Omron Sysmac Studio project 3.0_integration_v3 (Sysmac Studio 1.54.0.64019, StandardProject)

# Controller new_Controller_0: NJ301-1100 version 1.14
Units and slaves: Node1 : NX-ECC201 (E001); Unit 1 : NX-PC0020 (N1); Unit 2 : NX-ID5442 (N2); Unit 3 : NX-PC0010 (N3); Unit 4 : NX-PC0020 (N4); Unit 5 : NX-OD5121 (N5); Unit 6 : NX-PC0010 (N6); Power Supply : NJ-Px3001; CPU : NJ301-1100; 0 [Unit 0] : CJ1W-AD041-V1 (J01); 1 [Unit 1] : CJ1W-DA041 (J02); 2 : CJ1W-ID211 (J03); 3 : CJ1W-OC211 (J04)
Task PrimaryTask (priority 4, period or condition 1000): Program0

VAR_GLOBAL
    Station_1B2 : BOOL;  (* Branch 1 Extended; at IOBus://rack#0/slot#2/Ch1_In/Ch1_In05; published *)
    Station_1B1 : BOOL;  (* Branch 1 Retracted; at IOBus://rack#0/slot#2/Ch1_In/Ch1_In04; published *)
    Station_B4 : BOOL;  (* Slide Full; at IOBus://rack#0/slot#2/Ch1_In/Ch1_In03; published *)
    Station_3S1 : BOOL;  (* arm_in_magazine; published *)
    Station_3S2 : BOOL;  (* arm_in_downstream; published *)
    Station_2B1 : BOOL;  (* Branch 2 Retracted; at IOBus://rack#0/slot#2/Ch1_In/Ch1_In06; published *)
    Panel_S1 : BOOL;  (* start_button; at IOBus://rack#0/slot#2/Ch1_In/Ch1_In08; published *)
    Panel_S2 : BOOL;  (* stop_button; at IOBus://rack#0/slot#2/Ch1_In/Ch1_In09; published *)
    Panel_S4 : BOOL;  (* reset_button; at IOBus://rack#0/slot#2/Ch1_In/Ch1_In11; published *)
    Station_K1 : BOOL;  (* Conveyor Motor ON; at IOBus://rack#0/slot#3/Ch1_Out/Ch1_Out00; published *)
    Station_1Y1 : BOOL;  (* Branch 1 to extend; at IOBus://rack#0/slot#3/Ch1_Out/Ch1_Out01; published *)
    Station_2Y1 : BOOL;  (* Branch 2 extended; at IOBus://rack#0/slot#3/Ch1_Out/Ch1_Out02; published *)
    Station_3Y1 : BOOL;  (* Stopper to Retract; at IOBus://rack#0/slot#3/Ch1_Out/Ch1_Out03; published *)
    Station_3Y2 : BOOL;  (* arm_2_downstream; published *)
    Station_H1 : BOOL;  (* start light; at IOBus://rack#0/slot#3/Ch1_Out/Ch1_Out08; published *)
    Station_H2 : BOOL;  (* reset light; at IOBus://rack#0/slot#3/Ch1_Out/Ch1_Out09; published *)
    Panel_H3 : BOOL;  (* Q1 light; at IOBus://rack#0/slot#3/Ch1_Out/Ch1_Out10; published *)
    Panel_H4 : BOOL;  (* Q2 light; at IOBus://rack#0/slot#3/Ch1_Out/Ch1_Out11; published *)
    Station_1B1_in : BOOL;
    Station_2B2 : BOOL;  (* Branch 2 Extended; at IOBus://rack#0/slot#2/Ch1_In/Ch1_In07 *)
    Part_AV : BOOL;  (* Workpiece Available; at IOBus://rack#0/slot#2/Ch1_In/Ch1_In00 *)
    Station_B2 : BOOL;  (* Metallic Workpiece; at IOBus://rack#0/slot#2/Ch1_In/Ch1_In01 *)
    Station_B3 : BOOL;  (* Workpiece Not Black; at IOBus://rack#0/slot#2/Ch1_In/Ch1_In02 *)
    IP_N_FO : BOOL;  (* Station Occupied; at IOBus://rack#0/slot#3/Ch1_Out/Ch1_Out07 *)
END_VAR

PROGRAM Program0
VAR
    FB_Panel_1 : FB_Panel;
    run_mode : BOOL;
    stop_mode : BOOL;
    reset_mode : BOOL;
    FB_Actuator_T1_1 : FB_Actuator_T1;
    timer_t1 : TON;
    error_mode : BOOL;
    FB_Actuator_T2_1 : FB_Actuator_T2;
    Piston : RS;
    error_ejec : BOOL;
    extend_piston : BOOL;
    workpiece_ready_set : BOOL;
    flip_flop_1 : RS;
    workpiece_ready : BOOL;
    workpiece_picked_up : BOOL;
    wait_for_piston : TON;
    error_state : BOOL;
    error_suction : BOOL;
    error_t1 : BOOL;
    error_t2 : BOOL;
    rs1 : RS;
    rs2 : RS;
    rs3 : RS;
    e1 : BOOL;
    e2 : BOOL;
    e3 : BOOL;
    error_lift : BOOL;
    error_q2_out : BOOL;
    Station_h3 : BOOL;
    Station_h4 : BOOL;
    Control_station_3_1 : Control_Station_3;
    start_button : BOOL;
    Integrated_start : BOOL;
    stop_button : BOOL;
    reset_button : BOOL;
    integrated_stop : BOOL;
    SCADA_start : BOOL;
    SCADA_stop : BOOL;
    SCADA_reset : BOOL;
    FB_sender_1 : FB_Sender;
END_VAR
VAR_EXTERNAL
    Station_3S1 : BOOL;
    Panel_S2 : BOOL;
    Station_3Y2 : BOOL;
    Station_3S2 : BOOL;
    Panel_S1 : BOOL;
    Station_3Y1 : BOOL;
    Panel_S4 : BOOL;
    Station_H1 : BOOL;
    Station_H2 : BOOL;
    Panel_H4 : BOOL;
    Panel_H3 : BOOL;
    Station_1B2 : BOOL;
    Station_1B1 : BOOL;
    Station_1Y1 : BOOL;
    Station_2Y1 : BOOL;
    Station_2B1 : BOOL;
    Station_B4 : BOOL;
    Station_B2 : BOOL;
    Part_AV : BOOL;
    Station_B3 : BOOL;
    Station_2B2 : BOOL;
    Station_K1 : BOOL;
    IP_N_FO : BOOL;
END_VAR

(* Section Section0: ladder, written here as Structured Text *)

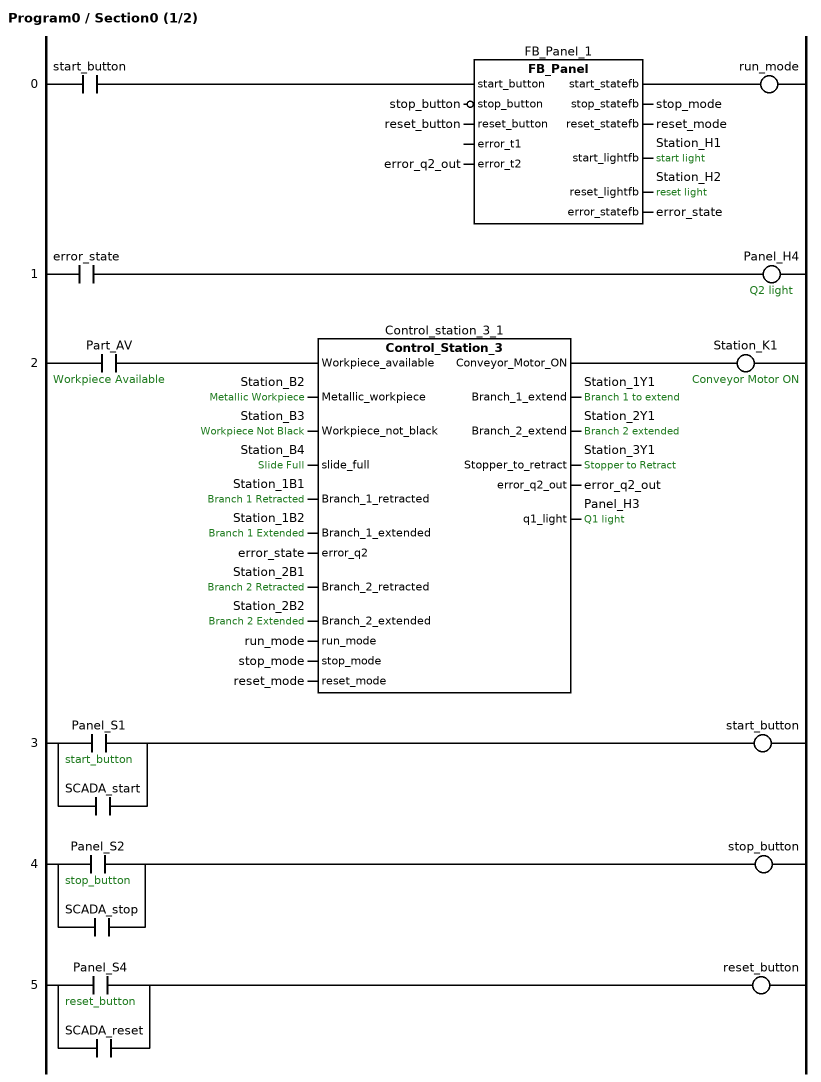
(* Rung 0 *)
FB_Panel_1(start_button := start_button, stop_button := NOT stop_button, reset_button := reset_button, error_t2 := error_q2_out, stop_statefb => stop_mode, reset_statefb => reset_mode, start_lightfb => Station_H1, reset_lightfb => Station_H2, error_statefb => error_state);
run_mode := FB_Panel_1.start_statefb;
(* Rung 1 *)
Panel_H4 := error_state;
(* Rung 2 *)
Control_station_3_1(Workpiece_available := Part_AV, Metallic_workpiece := Station_B2, Workpiece_not_black := Station_B3, slide_full := Station_B4, Branch_1_retracted := Station_1B1, Branch_1_extended := Station_1B2, error_q2 := error_state, Branch_2_retracted := Station_2B1, Branch_2_extended := Station_2B2, run_mode := run_mode, stop_mode := stop_mode, reset_mode := reset_mode, Branch_1_extend => Station_1Y1, Branch_2_extend => Station_2Y1, Stopper_to_retract => Station_3Y1, error_q2_out => error_q2_out, q1_light => Panel_H3);
Station_K1 := Control_station_3_1.Conveyor_Motor_ON;
(* Rung 3 *)
start_button := Panel_S1 OR SCADA_start;
(* Rung 4 *)
stop_button := Panel_S2 OR SCADA_stop;
(* Rung 5 *)
reset_button := Panel_S4 OR SCADA_reset;

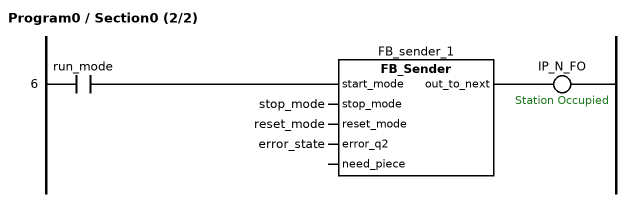
(* Rung 6 *)
FB_sender_1(start_mode := run_mode, stop_mode := stop_mode, reset_mode := reset_mode, error_q2 := error_state);
IP_N_FO := FB_sender_1.out_to_next;
END_PROGRAM

FUNCTION_BLOCK FB_Panel
VAR
    flip_flop : RS;
    flip_flop2 : RS;
    flip_flop_3 : RS;
    flip_flop3 : RS;
    stop_or_error : BOOL;
    error_q2 : BOOL;
    flip_flop4 : RS;
END_VAR
VAR_OUTPUT
    start_statefb : BOOL;
    stop_statefb : BOOL;
    reset_statefb : BOOL;
END_VAR
VAR_INPUT
    start_button : BOOL := False;
    stop_button : BOOL := False;
    reset_button : BOOL := False;
END_VAR
VAR_OUTPUT
    start_lightfb : BOOL;
    reset_lightfb : BOOL;
    error_statefb : BOOL;
END_VAR
VAR_INPUT
    error_t1 : BOOL;
    error_t2 : BOOL;
END_VAR
VAR_EXTERNAL
    Panel_H4 : BOOL;
END_VAR
(* ladder, written here as Structured Text *)

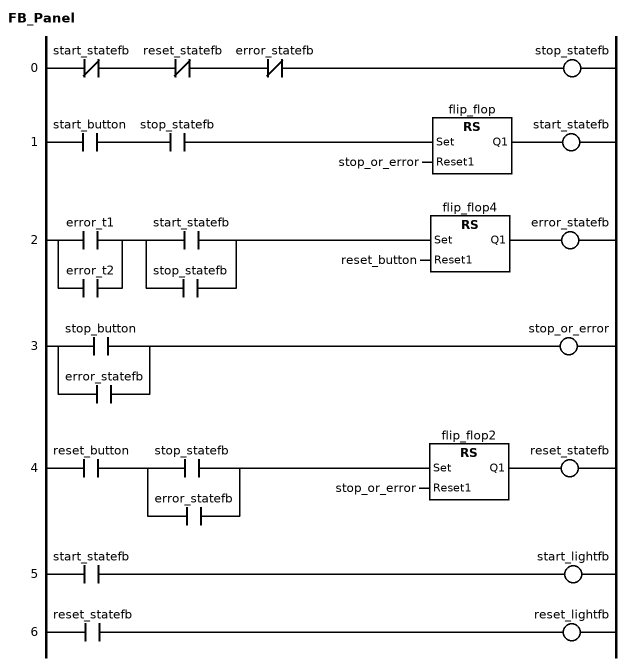
(* Rung 0 *)
stop_statefb := NOT start_statefb AND NOT reset_statefb AND NOT error_statefb;
(* Rung 1 *)
flip_flop(Set := start_button AND stop_statefb, Reset1 := stop_or_error);
start_statefb := flip_flop.Q1;
(* Rung 2 *)
flip_flop4(Set := (error_t1 OR error_t2) AND (start_statefb OR stop_statefb), Reset1 := reset_button);
error_statefb := flip_flop4.Q1;
(* Rung 3 *)
stop_or_error := stop_button OR error_statefb;
(* Rung 4 *)
flip_flop2(Set := reset_button AND (stop_statefb OR error_statefb), Reset1 := stop_or_error);
reset_statefb := flip_flop2.Q1;
(* Rung 5 *)
start_lightfb := start_statefb;
(* Rung 6 *)
reset_lightfb := reset_statefb;
END_FUNCTION_BLOCK

FUNCTION_BLOCK FB_Actuator_T1
VAR
    flip_flop_1 : RS;
    flip_flop_2 : RS;
    reset_to_home : BOOL;
    timer_t1 : TON;
    flip_flop_3 : RS;
    timer_t2 : TON;
    flip_flop_4 : RS;
    error_toSub : BOOL;
    error_toHome : BOOL;
    middle_timer : AccumulationTimer;
    flip_flop_5 : RS;
    reset_middle : BOOL;
    flip_flop6 : RS;
    move_to_middle_from_home : BOOL;
    move_to_home : BOOL;
    move_to_middle_from_sub : BOOL;
    unknown_pos : BOOL;
    reset_vac_arm_to_sub : BOOL;
    timer_t3 : TON;
    t : TIME;
    unknown_pos_timer : TON;
    TOF_1 : TOF;
    move_to_sub : BOOL;
END_VAR
VAR_INPUT
    Arm_In_Mag_Pos : BOOL;
    Arm_In_Sub_Pos : BOOL;
    stop_mode : BOOL;
END_VAR
VAR_OUTPUT
    error_arm : BOOL;
    arm_to_sub : BOOL;
    arm_to_home : BOOL;
END_VAR
VAR_INPUT
    error_q2 : BOOL;
    set_move_to_sub : BOOL;
    set_move_to_home : BOOL;
    set_move_to_middle_from_home : BOOL;
    set_move_to_middle_from_sub : BOOL;
END_VAR
VAR_OUTPUT
    middle_pos : BOOL;
END_VAR
VAR_INPUT
    reset_mode : BOOL;
END_VAR
VAR_EXTERNAL
    Station_1B1 : BOOL;
END_VAR
(* ladder, written here as Structured Text *)

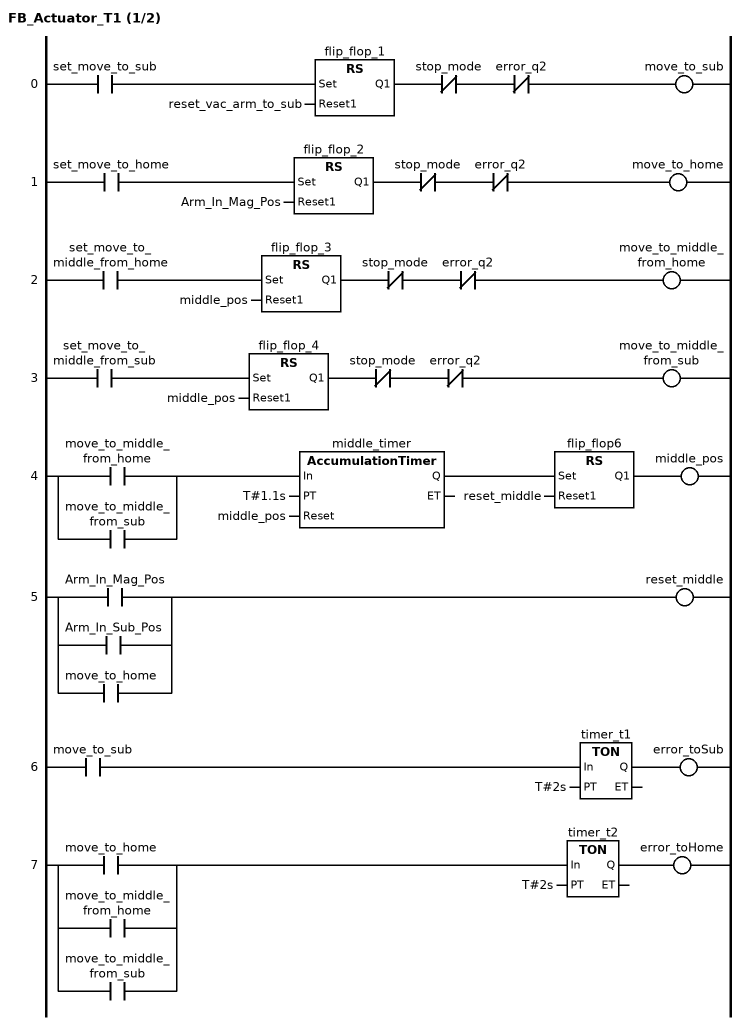
(* Rung 0 *)
flip_flop_1(Set := set_move_to_sub, Reset1 := reset_vac_arm_to_sub);
move_to_sub := flip_flop_1.Q1 AND NOT stop_mode AND NOT error_q2;
(* Rung 1 *)
flip_flop_2(Set := set_move_to_home, Reset1 := Arm_In_Mag_Pos);
move_to_home := flip_flop_2.Q1 AND NOT stop_mode AND NOT error_q2;
(* Rung 2 *)
flip_flop_3(Set := set_move_to_middle_from_home, Reset1 := middle_pos);
move_to_middle_from_home := flip_flop_3.Q1 AND NOT stop_mode AND NOT error_q2;
(* Rung 3 *)
flip_flop_4(Set := set_move_to_middle_from_sub, Reset1 := middle_pos);
move_to_middle_from_sub := flip_flop_4.Q1 AND NOT stop_mode AND NOT error_q2;
(* Rung 4 *)
middle_timer(In := move_to_middle_from_home OR move_to_middle_from_sub, PT := T#1.1s, Reset := middle_pos);
flip_flop6(Set := middle_timer.Q, Reset1 := reset_middle);
middle_pos := flip_flop6.Q1;
(* Rung 5 *)
reset_middle := Arm_In_Mag_Pos OR Arm_In_Sub_Pos OR move_to_home;
(* Rung 6 *)
timer_t1(In := move_to_sub, PT := T#2s);
error_toSub := timer_t1.Q;
(* Rung 7 *)
timer_t2(In := move_to_home OR move_to_middle_from_home OR move_to_middle_from_sub, PT := T#2s);
error_toHome := timer_t2.Q;

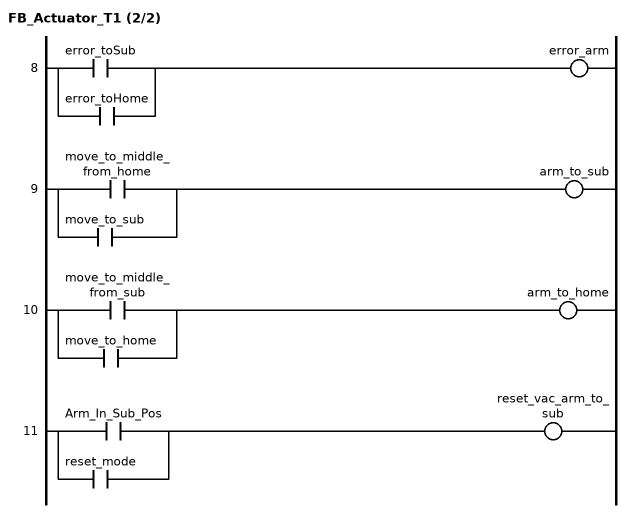
(* Rung 8 *)
error_arm := error_toSub OR error_toHome;
(* Rung 9 *)
arm_to_sub := move_to_middle_from_home OR move_to_sub;
(* Rung 10 *)
arm_to_home := move_to_middle_from_sub OR move_to_home;
(* Rung 11 *)
reset_vac_arm_to_sub := Arm_In_Sub_Pos OR reset_mode;
END_FUNCTION_BLOCK

FUNCTION_BLOCK Control_Station_3
VAR
    TON_workpiece_to_testing : TON;
    FB_Actuator_T2_1 : FB_Actuator_T2;
    ready_to_sort : BOOL;
    workpiece_counter : CTUD;
    workpiece_in_queue : BOOL;
    Stopper : FB_Actuator_T3;
    workpiece_passed : BOOL;
    cnt : INT;
    eject_magenta_rs : RS;
    eject_magenta : BOOL;
    eject_black : BOOL;
    eject_metallic : BOOL;
    one_block_through_stopper : TOF;
    extend_stopper : BOOL;
    eject_metallic_rs : RS;
    eject_black_rs : RS;
    reset_eject_magenta : BOOL;
    TON_reset_magenta : TON;
    TON_reset_metallic : TON;
    reset_eject_metallic : BOOL;
    TON_reset_black : TON;
    reset_eject_black : BOOL;
    TP_move_workpiece_to_test : TP;
    wait_at_test : TON;
    wait_at_test_2 : TON;
    Wait_at_test_3 : TON;
    move_workpiece_to_test : BOOL;
    sort_workpiece : BOOL;
    stopper_pulse : TP;
    close_workpiece : AccumulationTimer;
    arm_extended : BOOL;
    stopper_timer : AccumulationTimer;
    retract_stopper : BOOL;
    branch_1 : FB_Actuator_T2;
    reset_eject : BOOL;
    extend_branch_1_command : BOOL;
    retract_branch_1_command : BOOL;
    error_branch_1 : BOOL;
    branch_2 : FB_Actuator_T2;
    extend_branch_2_command : BOOL;
    retract_branch_2_command : BOOL;
    error_branch_2 : BOOL;
    add_to_counter : TON;
    CU_workpiece_counter : BOOL;
    queue_double_up_TON : TON;
    CU_double_up_counter : BOOL;
    rs_error_branch_2 : RS;
    test_error_branch_2 : BOOL;
    rs_error_branch_1 : RS;
    test_error_branch_1 : BOOL;
    set_reset_Branch_1_RS : RS;
    extend_branch_1 : BOOL;
    retract_branch_1 : BOOL;
    retract_branch_2 : BOOL;
    extend_branch_2 : BOOL;
    set_reset_Branch_2 : RS;
    double_up_queue_RS : RS;
    ET1 : TIME;
    reset_double_up : BOOL;
    queue_double_up_accTim : AccumulationTimer;
    ET : TIME;
    stop : BOOL;
    slide_full_TON : TON;
    slide_full_rs : RS;
    slide_full_error : BOOL;
    workpiece_removed_from_belt : AccumulationTimer;
    error_workpiece_removed : BOOL;
    black_slide_counter : CTU;
    metallic_slide_counter : CTU;
    magenta_slide_counter : CTU;
    black_cnt : INT;
    metallic_cnt : INT;
    magenta_cnt : INT;
    black_slide_full : BOOL;
    metallic_slide_full : BOOL;
    magenta_slide_full : BOOL;
    Delay_q2_branches : TON;
    branch_q2_error : BOOL;
END_VAR
VAR_INPUT
    Workpiece_available : BOOL;
    Metallic_workpiece : BOOL;
    Workpiece_not_black : BOOL;
    slide_full : BOOL;
    Branch_1_retracted : BOOL;
    Branch_1_extended : BOOL;
    error_q2 : BOOL;
    Branch_2_retracted : BOOL;
    Branch_2_extended : BOOL;
    run_mode : BOOL;
END_VAR
VAR_OUTPUT
    Conveyor_Motor_ON : BOOL;
    Branch_1_extend : BOOL;
    Branch_2_extend : BOOL;
    Stopper_to_retract : BOOL;
END_VAR
VAR_INPUT
    stop_mode : BOOL;
    reset_mode : BOOL;
END_VAR
VAR_OUTPUT
    error_q2_out : BOOL;
    q1_light : BOOL;
END_VAR
VAR_EXTERNAL
    Station_1B1 : BOOL;
    Station_1B1_in : BOOL;
    Station_1B2 : BOOL;
    Station_B2 : BOOL;
END_VAR
VAR
    _e1 : R_TRIG;
    _e2 : R_TRIG;
    _e3 : R_TRIG;
    _e4 : R_TRIG;
    _e5 : R_TRIG;
END_VAR
(* ladder, written here as Structured Text *)

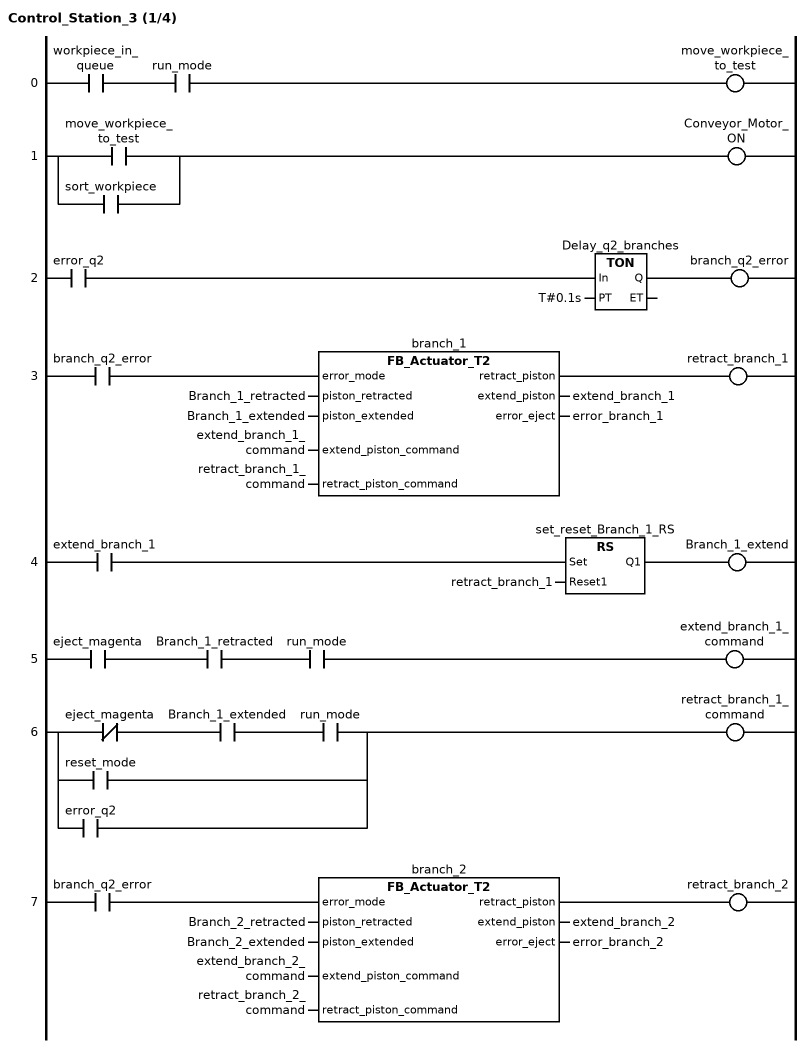
(* Rung 0 *)
move_workpiece_to_test := workpiece_in_queue AND run_mode;
(* Rung 1 *)
Conveyor_Motor_ON := move_workpiece_to_test OR sort_workpiece;
(* Rung 2 *)
Delay_q2_branches(In := error_q2, PT := T#0.1s);
branch_q2_error := Delay_q2_branches.Q;
(* Rung 3 *)
branch_1(error_mode := branch_q2_error, piston_retracted := Branch_1_retracted, piston_extended := Branch_1_extended, extend_piston_command := extend_branch_1_command, retract_piston_command := retract_branch_1_command, extend_piston => extend_branch_1, error_eject => error_branch_1);
retract_branch_1 := branch_1.retract_piston;
(* Rung 4 *)
set_reset_Branch_1_RS(Set := extend_branch_1, Reset1 := retract_branch_1);
Branch_1_extend := set_reset_Branch_1_RS.Q1;
(* Rung 5 *)
extend_branch_1_command := eject_magenta AND Branch_1_retracted AND run_mode;
(* Rung 6 *)
retract_branch_1_command := (NOT eject_magenta AND Branch_1_extended AND run_mode) OR reset_mode OR error_q2;
(* Rung 7 *)
branch_2(error_mode := branch_q2_error, piston_retracted := Branch_2_retracted, piston_extended := Branch_2_extended, extend_piston_command := extend_branch_2_command, retract_piston_command := retract_branch_2_command, extend_piston => extend_branch_2, error_eject => error_branch_2);
retract_branch_2 := branch_2.retract_piston;

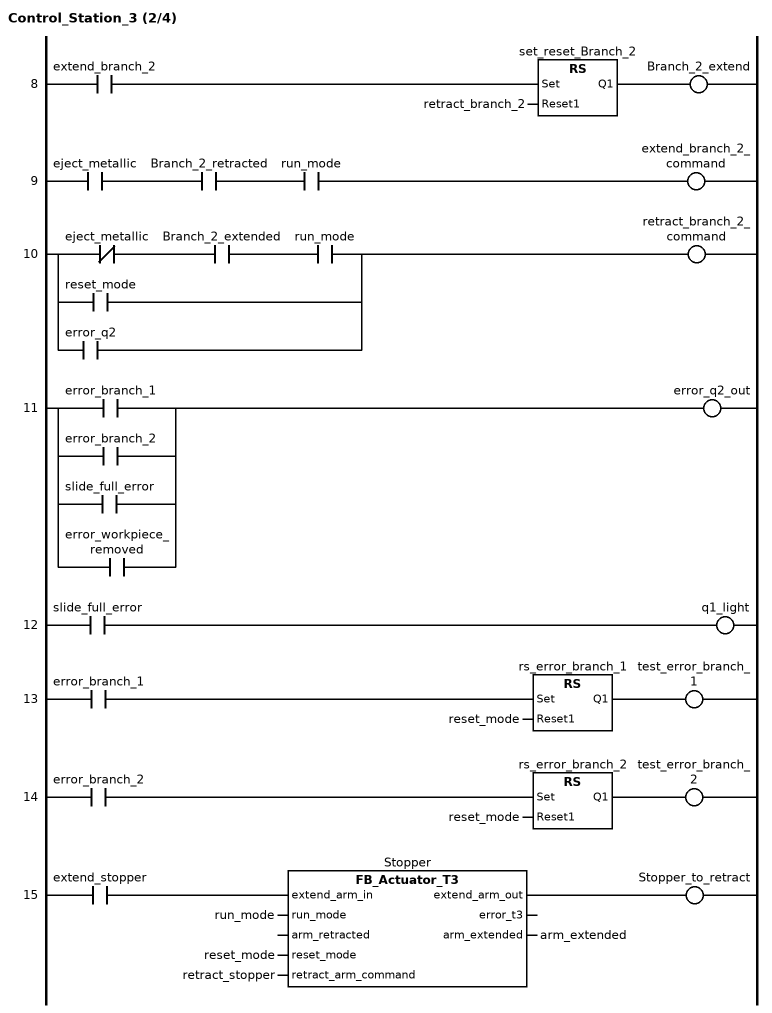
(* Rung 8 *)
set_reset_Branch_2(Set := extend_branch_2, Reset1 := retract_branch_2);
Branch_2_extend := set_reset_Branch_2.Q1;
(* Rung 9 *)
extend_branch_2_command := eject_metallic AND Branch_2_retracted AND run_mode;
(* Rung 10 *)
retract_branch_2_command := (NOT eject_metallic AND Branch_2_extended AND run_mode) OR reset_mode OR error_q2;
(* Rung 11 *)
error_q2_out := error_branch_1 OR error_branch_2 OR slide_full_error OR error_workpiece_removed;
(* Rung 12 *)
q1_light := slide_full_error;
(* Rung 13 *)
rs_error_branch_1(Set := error_branch_1, Reset1 := reset_mode);
test_error_branch_1 := rs_error_branch_1.Q1;
(* Rung 14 *)
rs_error_branch_2(Set := error_branch_2, Reset1 := reset_mode);
test_error_branch_2 := rs_error_branch_2.Q1;
(* Rung 15 *)
Stopper(extend_arm_in := extend_stopper, run_mode := run_mode, reset_mode := reset_mode, retract_arm_command := retract_stopper, arm_extended => arm_extended);
Stopper_to_retract := Stopper.extend_arm_out;

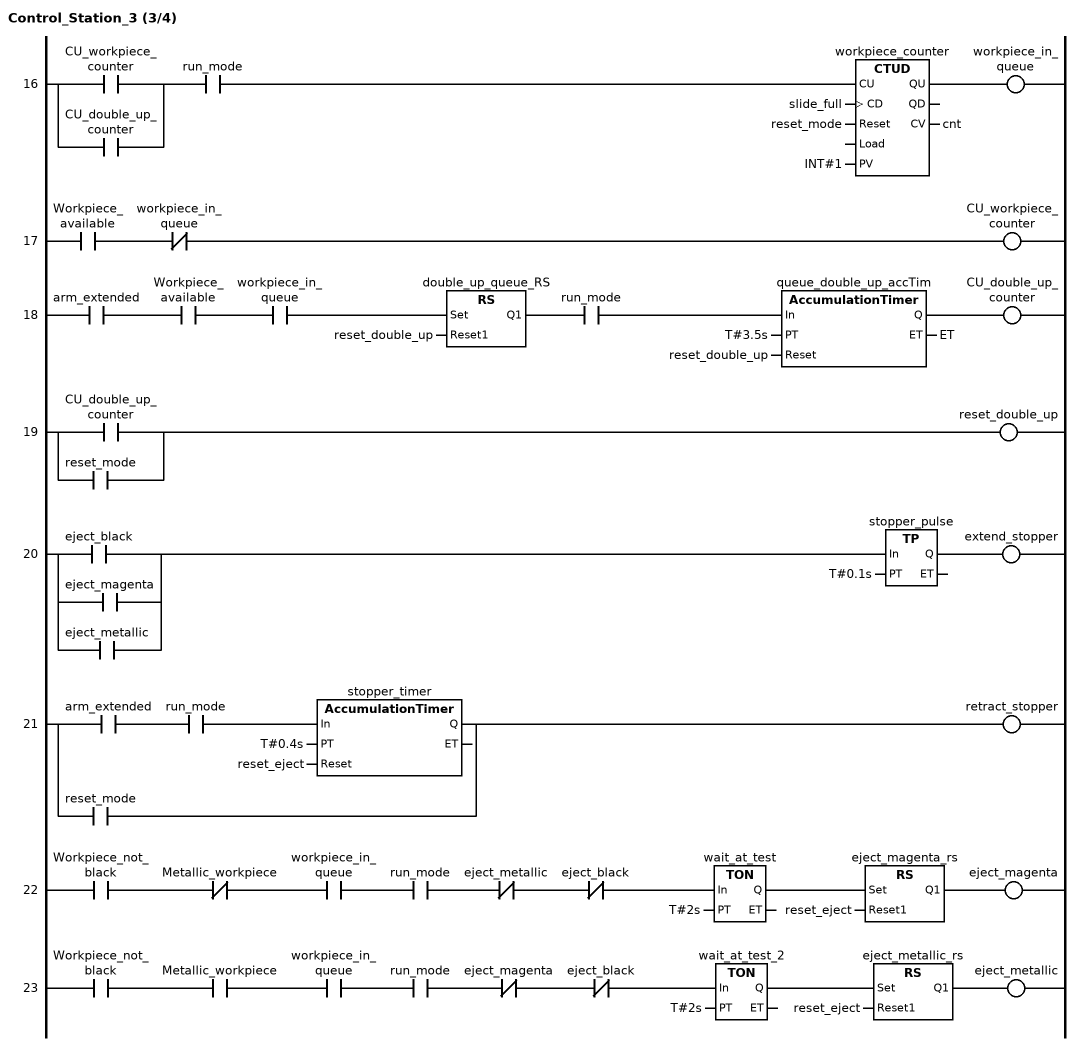
(* Rung 16 *)
_e1(CLK := slide_full);
_e2(CLK := (CU_workpiece_counter OR CU_double_up_counter) AND run_mode);
workpiece_counter(CU := _e2.Q, CD := _e1.Q, Reset := reset_mode, PV := INT#1, CV => cnt);
workpiece_in_queue := workpiece_counter.QU;
(* Rung 17 *)
CU_workpiece_counter := Workpiece_available AND NOT workpiece_in_queue;
(* Rung 18 *)
double_up_queue_RS(Set := arm_extended AND Workpiece_available AND workpiece_in_queue, Reset1 := reset_double_up);
queue_double_up_accTim(In := double_up_queue_RS.Q1 AND run_mode, PT := T#3.5s, Reset := reset_double_up, ET => ET);
CU_double_up_counter := queue_double_up_accTim.Q;
(* Rung 19 *)
reset_double_up := CU_double_up_counter OR reset_mode;
(* Rung 20 *)
stopper_pulse(In := eject_black OR eject_magenta OR eject_metallic, PT := T#0.1s);
extend_stopper := stopper_pulse.Q;
(* Rung 21 *)
stopper_timer(In := arm_extended AND run_mode, PT := T#0.4s, Reset := reset_eject);
retract_stopper := stopper_timer.Q OR reset_mode;
(* Rung 22 *)
wait_at_test(In := Workpiece_not_black AND NOT Metallic_workpiece AND workpiece_in_queue AND run_mode AND NOT eject_metallic AND NOT eject_black, PT := T#2s);
eject_magenta_rs(Set := wait_at_test.Q, Reset1 := reset_eject);
eject_magenta := eject_magenta_rs.Q1;
(* Rung 23 *)
wait_at_test_2(In := Workpiece_not_black AND Metallic_workpiece AND workpiece_in_queue AND run_mode AND NOT eject_magenta AND NOT eject_black, PT := T#2s);
eject_metallic_rs(Set := wait_at_test_2.Q, Reset1 := reset_eject);
eject_metallic := eject_metallic_rs.Q1;

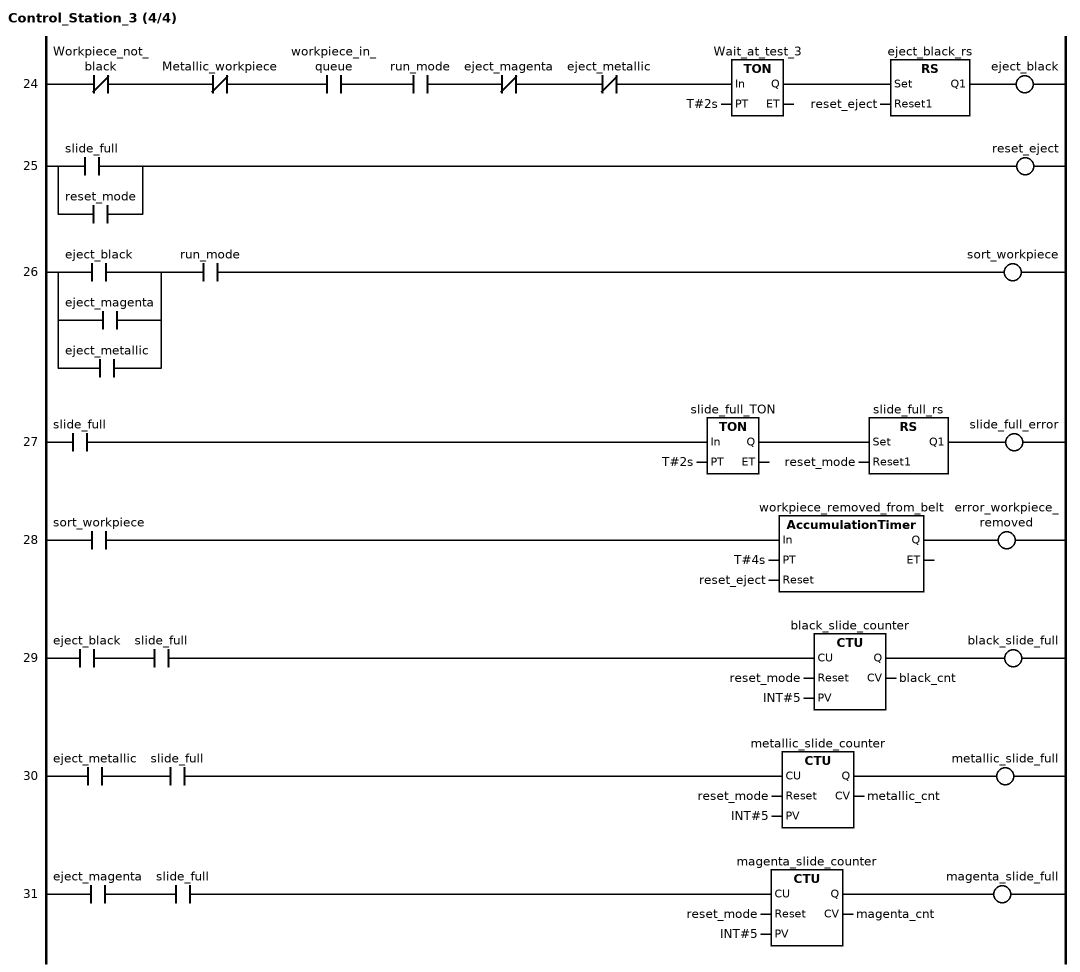
(* Rung 24 *)
Wait_at_test_3(In := NOT Workpiece_not_black AND NOT Metallic_workpiece AND workpiece_in_queue AND run_mode AND NOT eject_magenta AND NOT eject_metallic, PT := T#2s);
eject_black_rs(Set := Wait_at_test_3.Q, Reset1 := reset_eject);
eject_black := eject_black_rs.Q1;
(* Rung 25 *)
reset_eject := slide_full OR reset_mode;
(* Rung 26 *)
sort_workpiece := (eject_black OR eject_magenta OR eject_metallic) AND run_mode;
(* Rung 27 *)
slide_full_TON(In := slide_full, PT := T#2s);
slide_full_rs(Set := slide_full_TON.Q, Reset1 := reset_mode);
slide_full_error := slide_full_rs.Q1;
(* Rung 28 *)
workpiece_removed_from_belt(In := sort_workpiece, PT := T#4s, Reset := reset_eject);
error_workpiece_removed := workpiece_removed_from_belt.Q;
(* Rung 29 *)
_e3(CLK := eject_black AND slide_full);
black_slide_counter(CU := _e3.Q, Reset := reset_mode, PV := INT#5, CV => black_cnt);
black_slide_full := black_slide_counter.Q;
(* Rung 30 *)
_e4(CLK := eject_metallic AND slide_full);
metallic_slide_counter(CU := _e4.Q, Reset := reset_mode, PV := INT#5, CV => metallic_cnt);
metallic_slide_full := metallic_slide_counter.Q;
(* Rung 31 *)
_e5(CLK := eject_magenta AND slide_full);
magenta_slide_counter(CU := _e5.Q, Reset := reset_mode, PV := INT#5, CV => magenta_cnt);
magenta_slide_full := magenta_slide_counter.Q;
END_FUNCTION_BLOCK

FUNCTION_BLOCK FB_Actuator_T3
VAR
    TOF_1 : TOF;
    extend_arm_error_rs : RS;
    extend_arm_error_TON : TON;
    retract_arm : BOOL;
    Error_held_timer : AccumulationTimer;
    arm_extended_out : BOOL;
    reset_timer : BOOL;
    arm_out_timer : TON;
    arm_out_rs : RS;
    arm_extended_rs : RS;
    cycle_check_rs : RS;
    error_t3_1 : BOOL;
END_VAR
VAR_INPUT
    extend_arm_in : BOOL;
END_VAR
VAR_OUTPUT
    extend_arm_out : BOOL;
END_VAR
VAR_INPUT
    run_mode : BOOL;
    arm_retracted : BOOL;
END_VAR
VAR_OUTPUT
    error_t3 : BOOL;
END_VAR
VAR_INPUT
    reset_mode : BOOL;
    retract_arm_command : BOOL;
END_VAR
VAR_OUTPUT
    arm_extended : BOOL;
END_VAR
(* ladder, written here as Structured Text *)

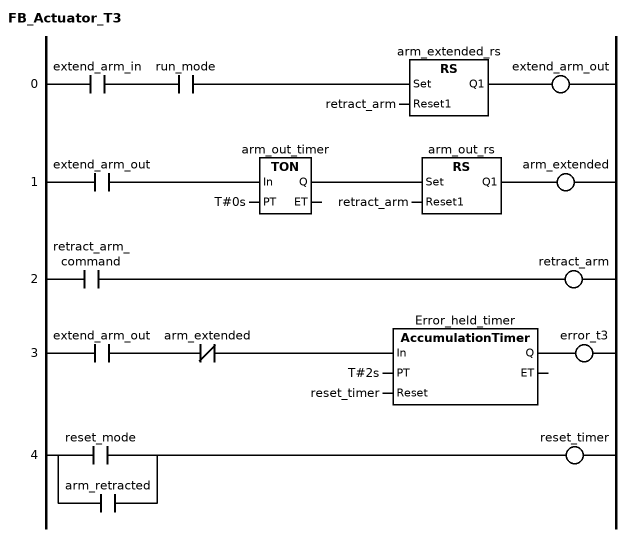
(* Rung 0 *)
arm_extended_rs(Set := extend_arm_in AND run_mode, Reset1 := retract_arm);
extend_arm_out := arm_extended_rs.Q1;
(* Rung 1 *)
arm_out_timer(In := extend_arm_out, PT := T#0s);
arm_out_rs(Set := arm_out_timer.Q, Reset1 := retract_arm);
arm_extended := arm_out_rs.Q1;
(* Rung 2 *)
retract_arm := retract_arm_command;
(* Rung 3 *)
Error_held_timer(In := extend_arm_out AND NOT arm_extended, PT := T#2s, Reset := reset_timer);
error_t3 := Error_held_timer.Q;
(* Rung 4 *)
reset_timer := reset_mode OR arm_retracted;
END_FUNCTION_BLOCK

FUNCTION_BLOCK control_T3
VAR
    FB_Actuator_T3_2 : FB_Actuator_T3;
    retract_arm : BOOL;
    arm_extended : BOOL;
END_VAR
VAR_INPUT
    run_mode : BOOL;
    arm_retracted : BOOL;
    reset_mode : BOOL;
END_VAR
VAR_OUTPUT
    error_t3 : BOOL;
    extend_arm_out : BOOL;
END_VAR
VAR_INPUT
    extend_arm_in : BOOL;
END_VAR
(* ladder, written here as Structured Text *)

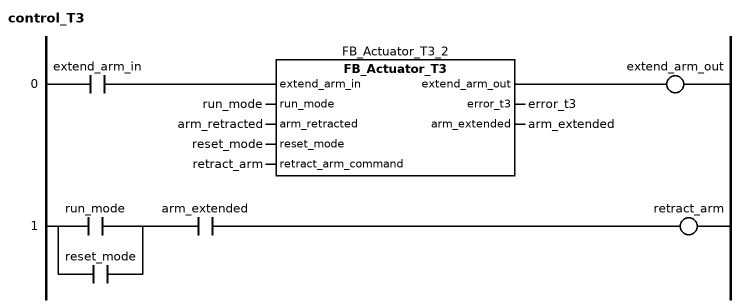
(* Rung 0 *)
FB_Actuator_T3_2(extend_arm_in := extend_arm_in, run_mode := run_mode, arm_retracted := arm_retracted, reset_mode := reset_mode, retract_arm_command := retract_arm, error_t3 => error_t3, arm_extended => arm_extended);
extend_arm_out := FB_Actuator_T3_2.extend_arm_out;
(* Rung 1 *)
retract_arm := (run_mode OR reset_mode) AND arm_extended;
END_FUNCTION_BLOCK

FUNCTION_BLOCK FB_Sender
VAR
    start_mode_pulse : BOOL;
    stop_mode_pulse : BOOL;
    reset_mode_pulse : BOOL;
    start_pulse : TP;
    stop_pulse : TP;
    reset_pulse : TP;
    T : TIME;
    np_pulse_t : TP;
    np_pulse : BOOL;
    TON_need_piece : TON;
    et1 : TIME;
    et2 : TIME;
    et3 : TIME;
    et4 : TIME;
    test_stop_pulse : AccumulationTimer;
    et5 : TIME;
    stop_signal_wait : BOOL;
    start_signal_wait : BOOL;
    reset_signal_wait : BOOL;
    stop_signal_TP : TP;
    start_signal_TP : TP;
    reset_signal_TP : TP;
    wait_need_piece : TON;
END_VAR
VAR_INPUT
    start_mode : BOOL;
    stop_mode : BOOL;
    reset_mode : BOOL;
    error_q2 : BOOL;
    need_piece : BOOL;
END_VAR
VAR_OUTPUT
    out_to_next : BOOL;
END_VAR
(* ladder, written here as Structured Text *)

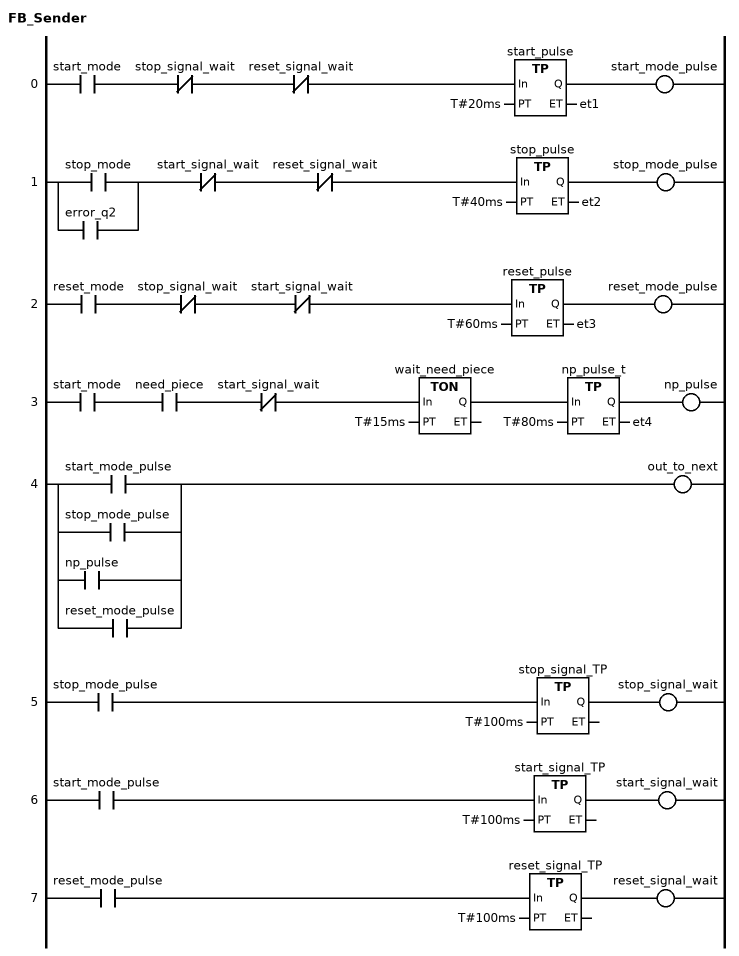
(* Rung 0 *)
start_pulse(In := start_mode AND NOT stop_signal_wait AND NOT reset_signal_wait, PT := T#20ms, ET => et1);
start_mode_pulse := start_pulse.Q;
(* Rung 1 *)
stop_pulse(In := (stop_mode OR error_q2) AND NOT start_signal_wait AND NOT reset_signal_wait, PT := T#40ms, ET => et2);
stop_mode_pulse := stop_pulse.Q;
(* Rung 2 *)
reset_pulse(In := reset_mode AND NOT stop_signal_wait AND NOT start_signal_wait, PT := T#60ms, ET => et3);
reset_mode_pulse := reset_pulse.Q;
(* Rung 3 *)
wait_need_piece(In := start_mode AND need_piece AND NOT start_signal_wait, PT := T#15ms);
np_pulse_t(In := wait_need_piece.Q, PT := T#80ms, ET => et4);
np_pulse := np_pulse_t.Q;
(* Rung 4 *)
out_to_next := start_mode_pulse OR stop_mode_pulse OR np_pulse OR reset_mode_pulse;
(* Rung 5 *)
stop_signal_TP(In := stop_mode_pulse, PT := T#100ms);
stop_signal_wait := stop_signal_TP.Q;
(* Rung 6 *)
start_signal_TP(In := start_mode_pulse, PT := T#100ms);
start_signal_wait := start_signal_TP.Q;
(* Rung 7 *)
reset_signal_TP(In := reset_mode_pulse, PT := T#100ms);
reset_signal_wait := reset_signal_TP.Q;
END_FUNCTION_BLOCK

FUNCTION_BLOCK FB_Actuator_T2
VAR
    reset_to_home : BOOL;
    retract_ff : RS;
    extend_ff : RS;
    extend_t : TON;
    retract_t : TON;
    retract_err : BOOL;
    extend_err : BOOL;
    workpiece_lifted : BOOL;
    Workpiece_ejection : RS;
END_VAR
VAR_OUTPUT
    retract_piston : BOOL;
END_VAR
VAR_INPUT
    error_mode : BOOL;
END_VAR
VAR_OUTPUT
    extend_piston : BOOL;
END_VAR
VAR_INPUT
    piston_retracted : BOOL;
    piston_extended : BOOL;
END_VAR
VAR_OUTPUT
    error_eject : BOOL;
END_VAR
VAR_INPUT
    extend_piston_command : BOOL;
    retract_piston_command : BOOL;
END_VAR
(* ladder, written here as Structured Text *)

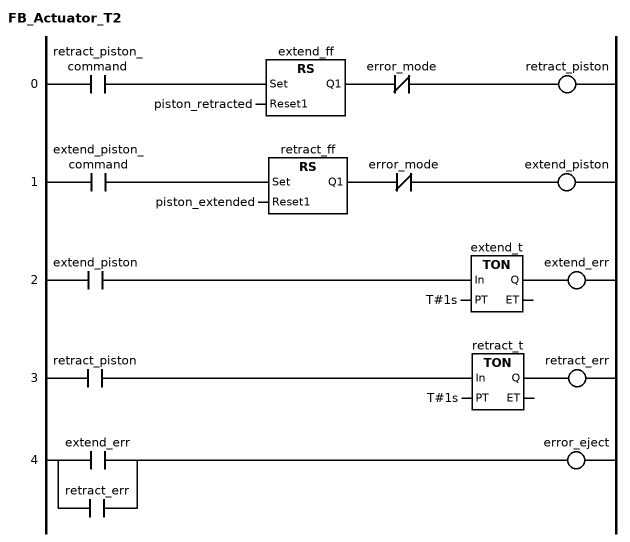
(* Rung 0 *)
extend_ff(Set := retract_piston_command, Reset1 := piston_retracted);
retract_piston := extend_ff.Q1 AND NOT error_mode;
(* Rung 1 *)
retract_ff(Set := extend_piston_command, Reset1 := piston_extended);
extend_piston := retract_ff.Q1 AND NOT error_mode;
(* Rung 2 *)
extend_t(In := extend_piston, PT := T#1s);
extend_err := extend_t.Q;
(* Rung 3 *)
retract_t(In := retract_piston, PT := T#1s);
retract_err := retract_t.Q;
(* Rung 4 *)
error_eject := extend_err OR retract_err;
END_FUNCTION_BLOCK